INTERFACE I_Collections

(* Number of elements in collection*)
PROPERTY _Count : DINT
GET
END_GET
END_PROPERTY

(* Gets collection's error status *)
PROPERTY _Error_Status : ST_ERROR
GET
END_GET
END_PROPERTY

(* Checks if collection is empty.*)
PROPERTY _Is_Empty : BOOL
GET
END_GET
END_PROPERTY

(* Empties/Clears/Deletes every element on the collection*)
METHOD Clear
END_METHOD

END_INTERFACE

(* stored: Version 1.1.0.1, ProductVersion 3.1.4024.4
   Itf I_Collections: Id {b40166ad-f1ab-4d22-a4d0-84895557404c}
   Property _Count: Id {23a45eae-6557-42b2-bda5-f817dab9f3d2}
   Get Get: Id {d366bad5-7796-4b69-a3d6-af0e937b23f0}
   Property _Error_Status: Id {be04b552-3c2b-4c54-a9e7-651f0a9a158f}
   Get Get: Id {eb2c4aed-dd87-4022-92be-3d474ee64a5e}
   Property _Is_Empty: Id {c45feb15-34b8-4188-816f-e2c0fc511e8c}
   Get Get: Id {66385950-96ba-40cb-ae27-099814d052ba}
   Method Clear: Id {3f8ee2bf-80ec-4210-a30e-6f79f6fe68c0} *)
